INTERFACE I_Members extends I_ListComponent

METHOD PUBLIC M_Abort : BOOL (* Return state complete*)
END_METHOD

METHOD PUBLIC M_Attach : BOOL
VAR_INPUT
	iParent:		I_Component;
	iComponent: 	I_Component;
END_VAR
END_METHOD

METHOD PUBLIC M_Detach : BOOL
VAR_INPUT
	iParent:	I_Component;
	iObject: 	I_Component;
END_VAR
END_METHOD

{attribute 'TcRpcEnable':='1'}
METHOD PUBLIC M_Mode : BOOL
VAR_INPUT
	eMode:		E_Mode;
END_VAR
END_METHOD

METHOD PUBLIC M_Reset : BOOL
END_METHOD

METHOD PUBLIC M_Start : BOOL (* Return state complete*)
END_METHOD

METHOD PUBLIC M_Stop : BOOL (* Return state complete*)
END_METHOD

{attribute 'OPC.UA.DA.Property' := '1'}
{attribute 'monitoring' := 'call'}
PROPERTY PUBLIC P_Length : DINT
GET
END_GET
END_PROPERTY

END_INTERFACE

(* stored: Version 1.1.0.1
   Itf I_Members: Id {2fbecd23-39f8-0ccf-3cc5-99cfd7eae8ff}
   Method M_Abort: Id {1f933af1-4f11-0ecb-08ec-82192c1a612b}
   Method M_Attach: Id {543e6ceb-65ee-0efc-1fe4-95b58138999e}
   Method M_Detach: Id {a56c8d05-9f85-03e8-06b4-d5828d4232ae}
   Method M_Mode: Id {771f8ed1-3d36-06da-31b9-43fac9a89313}
   Method M_Reset: Id {7335da18-63d0-00bd-1129-5875771dd0c7}
   Method M_Start: Id {66f0a26b-a021-0a30-25bb-222d89464134}
   Method M_Stop: Id {b825322c-1d24-0947-27e6-aec397e7e8ce}
   Property P_Length: Id {8a2135b4-d434-0b40-34a8-c68dbf9ce1b5}
   Get Get: Id {66a86cd6-d653-0b3d-1595-194313d1aca7} *)
